(* CoDeSys 2.3 export: INTERRUPT_0.EXP *)

(* POU Interrupt_0, ST *)
PROGRAM Interrupt_0
VAR
END_VAR
 %QX0.0 := 1;
END_PROGRAM
